RoboDK station: Init_SurgeryRobotics.rdk

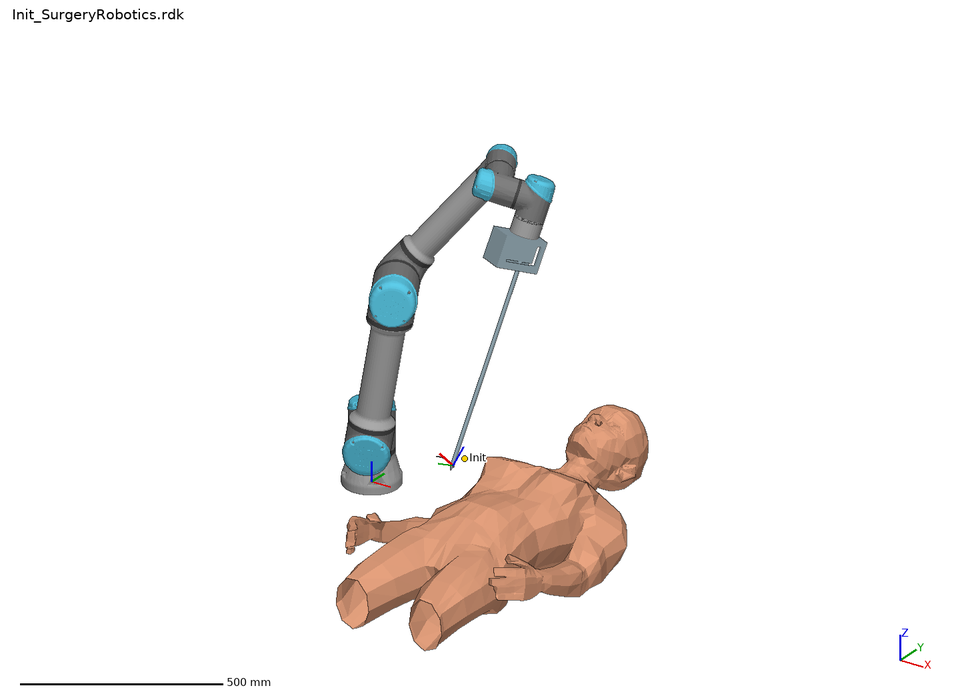
[picture v0: the station drawn from its stored meshes, robots at their saved joint values, targets as dots, program paths as lines]
Station Suture_solution (saved by RoboDK 5.9.0). Poses are relative to the parent item; angles as X-Y-Z fixed-axis rotations.
  - frame UR5e Base at (0, 0, 0) mm
    - robot UR5e: 6 axes, payload 5 kg, reach 850 mm, repeatability 0.03 mm, weight 18.4 kg
        modified DH rows (alpha deg, a mm, theta deg, d mm): 0, 0, 0, 162.5; 90, 0, 180, 0; 0, 425, 0, 0; 0, 392.25, 0, 133.3; -90, 0, 0, 99.7; 90, 0, 180, 99.6
        joint limits [-360, -360, -360, -360, -360, -360] to [360, 360, 360, 360, 360, 360]; home [0, -90, -90, 0, 90, 0]; saved at [30.678, -98.911, -31.325, -157.329, 76.626, -30.515]
      - tool Endowrist, TCP at (0, -15, 500) mm, rotated rx 180 ry 0 rz 0 deg, size 70 x 120 x 623 mm
        - frame Gripper at (0, 5, -105) mm, rotated rx 3.48 ry -10.1 rz -166.12 deg
          - object surgical_needle at (0, 0, 0) mm, size 47.8 x 42.3 x 2.9 mm, geometry from surgical_needle.obj
    - target Init (joint target) at (350, -100, 200) mm; joints [3.023, -79.004, -66.897, -124.099, 90, -86.977] of UR5e
    - object HumanBody1 at (0, 0, 0) mm, size 544.8 x 1046.4 x 300 mm, geometry from HumanBody1.obj
